{attribute 'call_after_init'}
FUNCTION_BLOCK AdsDataQueue
VAR
	elements : FB_BA_DynamicArray := (uiEntrySize := SIZEOF(POINTER TO AdsData), uiMinExpCount := CONSTS.initArraySize); 
	length : INT := 0;
	
	entrySize : UDINT;
END_VAR
(*
this container stores dynamically generated AdsData Structs
AdsData to be added are passed by reference, then this function block allocates a structure to be stored
AdsData are get() by reference and poll() by value
*)

METHOD clear : BOOL
VAR
	i : INT;
	temp : REFERENCE TO AdsData;
	tempAdr : POINTER TO AdsData;
END_VAR
FOR i:=0 TO length-1 BY 1 DO
	temp := get(index := i, getSize => );
	tempAdr := ADR(temp);
	__DELETE(tempAdr);
END_FOR

elements.Reset();
length := 0;
END_METHOD

METHOD contains : BOOL //check contents, not pointer value
VAR_INPUT
	value : REFERENCE TO AdsData;
END_VAR
VAR_OUTPUT
	atIndex : INT;
END_VAR
VAR
	temp : REFERENCE TO AdsData;
	i : INT;
END_VAR
IF length = 0 THEN
	contains := FALSE;
	RETURN;
END_IF

FOR i:=0 TO length-1 BY 1 DO
	temp := get(index := i, getSize => );
	
	IF 
		SIZEOF(value) = entrySize AND //same size
		MEMCMP(ADR(temp), ADR(value), SIZEOF(entrySize)) = 0 //same data
	THEN
		contains := TRUE;
		atIndex := i;
		RETURN;
	END_IF
	
END_FOR
contains := FALSE;
END_METHOD

METHOD get : REFERENCE TO AdsData
VAR_INPUT
	index : INT;
END_VAR
VAR_OUTPUT
	getSize : UDINT;
END_VAR
IF length = 0 OR index < 0 OR index >= length THEN
	getSize := 0;
ELSE
	elements.GetEntry(diIndex := index, pResultEntry := ADR(get));
	getSize := SIZEOF(get);
END_IF
END_METHOD

METHOD isEmpty : BOOL
VAR_INPUT
END_VAR
isEmpty := length = 0;
END_METHOD

METHOD poll : AdsData
VAR_OUTPUT
	getSize : UDINT;
END_VAR
IF length > 0 THEN
	poll := get(index := 0, getSize => getSize);
	elements.RemoveEntry(diIndex := 0);
	
	length := length - 1;
END_IF
END_METHOD

METHOD push : BOOL
VAR_INPUT
	value : REFERENCE TO AdsData;
END_VAR
VAR
	temp : POINTER TO AdsData;
END_VAR
temp := __NEW(AdsData);
temp^ := value;

elements.AddEntryPtr(pEntry := temp);

length := length + 1;
END_METHOD

METHOD set : BOOL
VAR_INPUT
	i : INT;
	value : REFERENCE TO AdsData;
END_VAR
VAR
	temp : REFERENCE TO AdsData;
END_VAR
IF length = 0 THEN
	RETURN;
END_IF

IF i >= 0 AND i < length THEN
	temp REF= get(i);
	temp := value;
	
	set := TRUE;
END_IF
END_METHOD

{attribute 'call_after_init'}
METHOD setup : BOOL
VAR_INPUT
END_VAR
entrySize := SIZEOF(AdsData);
END_METHOD

METHOD size : INT
size := length;
END_METHOD

END_FUNCTION_BLOCK

(* stored: Version 1.1.0.1, ProductVersion 3.1.4024.11
   POU AdsDataQueue: Id {31555f0d-7c4f-4350-b3a4-ff1b5982d4dd}, SpecialFunc None
   Method clear: Id {db44bf77-29ba-44a4-b4b0-ab8e1f12b8c0}
   Method contains: Id {a3bbf896-9f8a-48ee-84b2-aeaeb529bc15}
   Method get: Id {217c607c-584c-47a6-bd6b-45b399a5afab}
   Method isEmpty: Id {9a77362f-d3ac-4821-a848-453c2a700378}
   Method poll: Id {2750ad6b-3a36-4b2f-96d7-5f4c37362aba}
   Method push: Id {2868282b-9ddd-4f98-bf42-e70797839065}
   Method set: Id {581121c0-b6ec-4618-813a-c1cf00207d6e}
   Method setup: Id {efba3dbc-737b-427d-a6d2-60b710fa693f}
   Method size: Id {0fa383f9-597d-49f8-9fce-9ad607a5f6e6} *)
